{attribute 'GeneratedUsingTerminal: ELX3351-0000-0016'}
{attribute addProperty BoxType "ELX3351-0000-0016"}
{attribute addProperty Id "CtrlAT %Q*Ctrl_AEDC374E4"}
{attribute addProperty CRC "1234677494"}
{attribute addProperty Size "4"}
TYPE RMB_Control_4997AEF6 EXTENDS OutputBase_10CEE7DE :
STRUCT
	{attribute addProperty Name "Ctrl"}
	Ctrl AT %Q* : Ctrl_AEDC374E;
END_STRUCT
END_TYPE

(* stored: Version 1.2.0.0, ProductVersion 3.1.4024.9
   DUT RMB_Control_4997AEF6: Id {c1a710c3-3919-4190-a400-75b4ae737a63} *)
